FUNCTION_BLOCK FB_EnableAxis
VAR_INPUT
	bEnable			: BOOL;	(*Enable controller*)
	bHalt			: BOOL;	(*Halt stops the axis*)
	bReset			: BOOL;	(*Resets the controller*)
	wStatus			: WORD;	(*Status Word of the Controller*)

	bEnablePos		: BOOL;	(*Positive movement enabled*)
	bEnableNeg		: BOOL;	(*Negative movement enabled*)
	Override 		: LREAL;	(*Override for the axis*)
END_VAR
VAR_OUTPUT
	bDriveEnabled	: BOOL;	(*Controller is enabled*)
	bFaultActive	: BOOL;	(*Fault is active on controller*)
	wControl		: WORD;	(*Control word to Controller*)
END_VAR
VAR_IN_OUT
	AxisRef			: AXIS_REF;
END_VAR
VAR
	mcPower			: MC_Power;
	mcReset			: MC_Reset;
	fbEPOSControl	: FB_EPOS_Control;
	fb_Epos_SetEnabled: FB_SetEnableState;
END_VAR

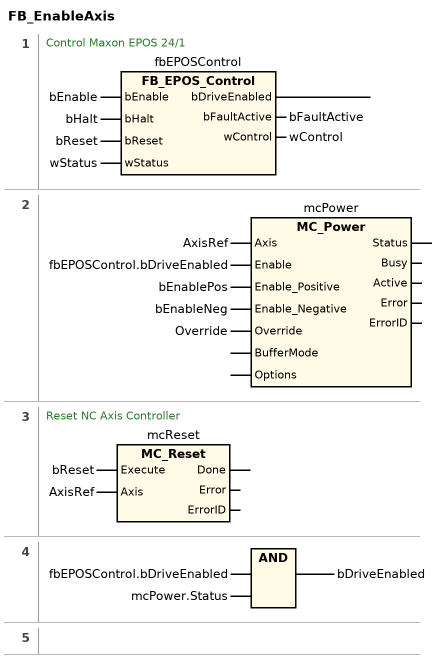
// NETWORK 1
// Control Maxon EPOS 24/1
fbEPOSControl(
    bEnable := bEnable,
    bHalt := bHalt,
    bReset := bReset,
    wStatus := wStatus,
    bFaultActive => bFaultActive,
    wControl => wControl); // FB_EPOS_Control

// NETWORK 2
mcPower(
    Axis := AxisRef,
    Enable := fbEPOSControl.bDriveEnabled,
    Enable_Positive := bEnablePos,
    Enable_Negative := bEnableNeg,
    Override := Override); // MC_Power

// NETWORK 3
// Reset NC Axis Controller
mcReset(Execute := bReset, Axis := AxisRef); // MC_Reset

// NETWORK 4
bDriveEnabled := fbEPOSControl.bDriveEnabled AND mcPower.Status;

// NETWORK 5

END_FUNCTION_BLOCK

(* stored: Version 1.1.0.1, ProductVersion 3.1.4024.2
   POU FB_EnableAxis: Id {7646a294-1942-442f-b4a3-3669063f84db}, SpecialFunc None *)
